PROGRAM MAIN
VAR

	nState: INT;

END_VAR


(*Setup a database  -  In that database make a table using this command in the Sql Query Editor...

CREATE TABLE `MyTable_Struct` 
(
	`ID` BIGINT NOT NULL AUTO_INCREMENT, 
	 `Timestamp` DATETIME, 
	 `Name` VARCHAR(80), 
	 `nSensor1` DOUBLE, 
	 `nSensor2` DOUBLE,

	 PRIMARY KEY (ID)
)

*)

CASE nState OF
	
0: //Idle

1: //DB write
	pWriteDB();
	IF NOT GVL.fbPLCDBWrite.bBusy THEN
		
		IF NOT GVL.fbPLCDBWrite.bError THEN
			nState := 2;
			ELSE
			nState := 3;
		END_IF;
	END_IF
	
2: //DB read
	pReadDB();
	IF NOT GVL.fbPLCDBRead.bBusy  THEN

		IF NOT GVL.fbPLCDBRead.bError THEN
			nState := 0;
			ELSE
			nState := 3;
		END_IF;
	END_IF;
	
3: //Error state


END_CASE

END_PROGRAM

(* stored: Version 1.1.0.1, ProductVersion 3.1.4024.9
   POU MAIN: Id {a9a1e98d-05c8-4d49-a39c-a97cbfea2453}, SpecialFunc None *)
